(* PLC project kneading, Dassault Systèmes ControlBuild 2024x *)
(* stored: creationDateTime 2023-10-03T11:13:38-01:00 *)

FUNCTION_BLOCK batch.kneading
  VAR_INPUT
    kneadingRequest : BOOL := false;
    cycleInProgress : BOOL := false;
    mixtureLevel : DINT := 0;
  END_VAR
  VAR_OUTPUT
    kneadingOK : BOOL := false;
  END_VAR
  VAR_OUTPUT
    knead : BOOL := false;
    clean : BOOL := false;
    cleaningEnd : BOOL := false;
    evacuateMixture : BOOL := false;
    evacMixtureEnd : BOOL := false;
  END_VAR
  VAR
    nbCycles : DINT := 0;
  END_VAR
  VAR CONSTANT
    kneadingDuration : DINT := 20;
    nbOfCleanCycles : DINT := 10;
    cleaningDuration : DINT := 30;
  END_VAR

INITIAL_STEP 10:
  10_INLINE1(N);
  COMPUTE_FUNCTION_BLOCKS(S);
END_STEP
ACTION 10_INLINE1:
  nbCycles := 0;
END_ACTION
TRANSITION FROM 10 TO 11
  := cycleInProgress;
END_TRANSITION
STEP 11:
END_STEP
TRANSITION FROM 11 TO 12
  := cycleInProgress AND kneadingRequest;
END_TRANSITION
STEP 12:
  12_INLINE2(N);
END_STEP
ACTION 12_INLINE2:
  knead;
END_ACTION
TRANSITION FROM 12 TO 13
  := NOT kneadingRequest;
END_TRANSITION
STEP 13:
  13_INLINE3(N);
END_STEP
ACTION 13_INLINE3:
  knead;
END_ACTION
TRANSITION FROM 13 TO 14
  := T/X13/kneadingDuration s;
END_TRANSITION
STEP 14:
  14_INLINE4(N);
END_STEP
ACTION 14_INLINE4:
  evacuateMixture;
END_ACTION
TRANSITION FROM 14 TO 15
  := mixtureLevel <= 1;
END_TRANSITION
STEP 15:
  15_INLINE5(N);
END_STEP
ACTION 15_INLINE5:
  IF(RE X15) THEN
  	nbCycles := nbCycles + 1;
  END_IF;
END_ACTION
TRANSITION FROM 15 TO 17
  := nbCycles < nbOfCleanCycles;
END_TRANSITION
TRANSITION FROM 15 TO 16
  := nbCycles >= nbOfCleanCycles;
END_TRANSITION
STEP 16:
  16_INLINE6(N);
END_STEP
ACTION 16_INLINE6:
  clean;
  knead;
  nbCycles := 0;
END_ACTION
TRANSITION FROM 16 TO 17
  := T/X16/cleaningDuration s;
END_TRANSITION
STEP 17:
  17_INLINE7(N);
END_STEP
ACTION 17_INLINE7:
  kneadingOK;
END_ACTION
TRANSITION FROM 17 TO 11
  := T/X17/500ms;
END_TRANSITION
ACTION COMPUTE_FUNCTION_BLOCKS:  (* blocks drawn on the SFC sheet *)
  G1:
END_ACTION

ACTION PostSFC:
IF NOT cycleInProgress THEN
	knead := FALSE;
	clean := FALSE;
	evacuateMixture := FALSE;
END_IF;

cleaningEnd := NOT cycleInProgress OR NOT clean;
evacMixtureEnd := NOT cycleInProgress OR NOT evacuateMixture;
END_ACTION
END_FUNCTION_BLOCK
